Staubli VAL3: Key_ListMC.pgx

program Key_ListMC(bool& x_bRefresh, num& x_nKeyValue, num& x_nSelectItem, num& x_nText)
begin

 call Key_ListBase(x_bRefresh,x_nKeyValue,x_nSelectItem)
  if x_bRefresh
     x_nText=0
    return
  endIf

    x_bRefresh=true
    switch x_nKeyValue
    //向左
    case 264
      x_nText=min(max(0,x_nText-1),2)
    break
    //向右
    case 268
      x_nText=max(min(2,x_nText+1),0)
    break

    default
      x_bRefresh=false
    break

    endSwitch




end
